(* POU Simulation/FB_Simu_Manipulator, ST *)
FUNCTION_BLOCK FB_Simu_Manipulator
(*Simulation model for the behaviour of the Manipulator.
Author: Niko Siltala, niko.siltala@tut.fi, Tampere University of Technology / MEI
Date: 2016-12-12
Version: 1.0
*)
VAR_INPUT
	bEnable			: BOOL := TRUE;	(*Enable manipulator*)
	bLift_Start		: BOOL;	(*Triggers and starts the lift movement at rising edge*)
	fLift_Velo		: REAL := 10;	(*Velocity*)
	fLift_TargetPos	: REAL;	(*Target position*)
	bBeam_Left		: BOOL;	(*Turn beam at left*)
	bBeam_Right		: BOOL;	(*Turn beam at right*)
	bGripper_Close	: BOOL; (*Close Gripper*)
END_VAR
VAR_OUTPUT
	bGripperIsOpen	: BOOL;	(*Gripper is open*)
	bLift_InTarget	: BOOL;	(*Lift has reached the target*)
	fLift_CurrentPos	: REAL;	(*Current position of the lift*)
	bLimit_Top		: BOOL;	(*Height position at top limit*)
	bLimit_Bottom	: BOOL;	(*Height position at bottom limit*)
	bHome_Sensor	: BOOL;	(*Height position at home limit*)
	bBeamAtRight	: BOOL;	(*Beam turned into right limit*)
	bBeamAtLeft		: BOOL;	(*Beam turned into left limit*)
END_VAR
VAR_IN_OUT
	stPart_inGripper : ST_Part; 	(*Data structure for the part*)
END_VAR
VAR
	fPos_angle	: REAL := 70;	(*Angle of beam [deg]*)
	fPos_height	: REAL;	(* Manipulators height position*)
	fPos_X		: REAL;	(* Manipulator's X position*)
	fPos_Y		: REAL;	(* Manipulator's Y position*)
	fBasePos_Y 	: REAL; (*Position of manipulator base*)
	iState_Lift		: UINT;	(*State of beam model*)
	fPos_Beam_L	: REAL;	(*Beam position left end*)
	fPos_Beam_R	: REAL;	(*Beam position right end*)
	bGripperClosed	: BOOL; (*Gripper is closed*)
	fPosFingerDiff 	: REAL;	(*Right finger position. 0 poistion when grasping.*)
	bInitDone		: BOOL;		(*Initialisation done for simulated machine*)
END_VAR
VAR CONSTANT
	iBEAM_LENGTH	: USINT := 120;	(*length of the beam*)
	fPOS_MAX_DOWN	: REAL	:= 220;	(*Max position for down movement*)
END_VAR
(*Simulate axis*)
IF NOT bEnable THEN
	iState_Lift := 0;
END_IF;

(*Initialisation*)
IF NOT bInitDone THEN
	(*Randomize system's starting position*)
	lastRandom := RDM(lastRandom);
	fLift_CurrentPos := -100 * lastRandom + 10;
	lastRandom := RDM(lastRandom);
	fPos_angle := 100 * lastRandom + 40; (* X2 = (180 - 100[=X1]) / 2 *)
	bInitDone:=TRUE;
END_IF;

CASE iState_Lift OF
0:	(*Off*)
	IF bEnable THEN
		iState_Lift := 1;
	ELSE
		bLift_InTarget := FALSE;
	END_IF;

1:	(*IDLE*)
	IF bLift_Start THEN
		bLift_InTarget := FALSE;
		iState_Lift := 2;
	END_IF;

2:	(*MovingToTarget*)
	bLift_InTarget := FALSE;
	IF fLift_TargetPos > fLift_CurrentPos THEN
		(*Moving up*)
		fLift_CurrentPos := fLift_CurrentPos + ABS(fLift_Velo);
	ELSIF fLift_TargetPos < fLift_CurrentPos THEN
		(*Moving down*)
		fLift_CurrentPos := fLift_CurrentPos - ABS(fLift_Velo);
	END_IF;
	(*Limit output*)
	fLift_CurrentPos := LIMIT(-220, fLift_CurrentPos, 10);
	(* Moved close to target*)
	IF (ABS(fLift_CurrentPos - fLift_TargetPos) <= ABS(fLift_Velo) ) THEN
		fLift_CurrentPos := fLift_TargetPos;
		iState_Lift := 3;
	END_IF;
	(*Start has been removed*)
	IF NOT bLift_Start THEN
		iState_Lift := 1;
	END_IF;

3:	(*In target*)
	bLift_InTarget := TRUE;
	IF NOT bLift_Start THEN
		iState_Lift := 1;
	END_IF;

ELSE	(*Error / to Default*)
	iState_Lift := 0;
END_CASE;

fPos_Y := -fLift_CurrentPos;


(*Simulate Beam turning*)
IF bBeam_Left AND (fPos_angle > 0) AND NOT bBeam_Right THEN
	fPos_angle := LIMIT(0, (fPos_angle - 15), 180);
END_IF;
IF bBeam_Right AND (fPos_angle < 180) AND NOT bBeam_Left THEN
	fPos_angle := LIMIT(0, (fPos_angle + 15), 180);
END_IF;


(*Calculate visualisation positions for lift and beam*)
fPos_X := -iBEAM_LENGTH*COS(3.1415926535897932384626433832795/180*fPos_angle);
(*fPos_Y := fPos_height;*)
fBasePos_Y := fPos_Y;	(*Used for animations as base position*)

(*Calculate endpositions of the visualisation for the beam*)
IF (fPos_X > 0) THEN
	fPos_Beam_L := 0;
	fPos_Beam_R := fPos_X;
ELSE
	fPos_Beam_L := fPos_X;
	fPos_Beam_R := 0;
END_IF;

(*define finger positions*)
IF bGripper_Close THEN
	fPosFingerDiff := 0;
ELSE
	fPosFingerDiff := 10;
END_IF;

(*Set sensor values*)
(*Set output values*)
bLimit_Top := (fPos_Y <= 0);
bLimit_Bottom := (fPos_Y >= 210);
bHome_Sensor := (fPos_Y <= 5) AND (fPos_Y >= -5);

bBeamAtLeft := (fPos_angle <= 0);
bBeamAtRight := (fPos_angle >= 180);

bGripperIsOpen := NOT bGripper_Close;
bGripperClosed := bGripper_Close;
END_FUNCTION_BLOCK

(* POU Simulation/RDM_From_OSCAT/RDM, ST *)
FUNCTION RDM : REAL
VAR_INPUT
	last : REAL;
END_VAR
VAR
	tn : DWORD;
	tc : INT;
END_VAR
(*
FROM OSCAT 333
version 1.9	10. mar. 2009
programmer 	hugo
tested by		tobias

this function calculates a pseudo random number
to generate the number it reads the sps timer and calculates a random number between 0 and 1:
in order to use rdm more then once within one sps cycle it need to be called with different seed numbers LAST.

*)
tn := T_PLC_MS();
tc := BIT_COUNT(tn);
tn.31 := tn.2;
tn.30 := tn.5;
tn.29 := tn.4;
tn.28 := tn.1;
tn.27 := tn.0;
tn.26 := tn.7;
tn.25 := tn.6;
tn.24 := tn.3;
tn := ROL(tn,BIT_COUNT(tn)) OR 16#80000001;
tn := tn MOD 71474513 + INT_TO_DWORD(tc + 77);
RDM := FRACT(DWORD_TO_REAL(tn) / 10000000.0 * (math.E - LIMIT(0.0,last,1.0)));


(*
pt := ADR(temp);
pt^ := (T_PLC_MS() AND 16#007FFFFF) OR 16#3D000000;
RDM := fract(modR(temp*e+pi1, PI1-last) + modR(temp*PI1+e + last,e-last));
*)

(* revision history
hm		16. jan 2007		rev 1.0
	original version

hm		11. nov 2007		rev 1.1
	changed time() into t_plc_ms()

hm		20. nov 2007		rev 1.2
	changed code of temp calculation to avoid overflow in modr due to resuclt would not fit DINT for high timeer values

hm		5. jan 2008		rev 1.3
	changed calculation of temp to avoid problem with high values of t_plc_ms

hm		2. feb 2008		rev 1.4
	changed algorithm to avoind non iec functions and guarantee more randomness

hm	10. mar. 2008		rev 1.5
	make sure last will be between 0 and 1 to avoid invalid results

hm	16. mar. 2008		rev 1.6
	added conversion for tc to avoid warnings under codesys 3.0

hm	18. may. 2008		rev 1.7
	changed constant E to E1

hm	18. oct. 2008		rev 1.8
	using math constants

hm	10. mar. 2009		rev 1.9
	real constants updated to new systax using dot

*)
END_FUNCTION

(* POU Simulation/RDM_From_OSCAT/T_PLC_MS, ST *)
FUNCTION T_PLC_MS : DWORD
VAR CONSTANT
	debug : BOOL := 0;
	N : INT := 0;
	offset : DWORD := 0;
END_VAR
VAR
	tx : TIME;
END_VAR
(*
	From OSCAT 333
	version 1.2	16. nov 2008
	programmer 	hugo
	tested BY	oscat

	T_PLC_MS reads the internal PLC timer AND RETURN the TIME, it has the advantage TO be able TO set a debug mode
AND SPEED up the counter TO test the plc timer overrun which occurs every 50 days respectively 25 days AT siemens S7
	this routine also allows TO correct the behavior OF s7 where the internal plc counter will NOT count all 32 bits.
*)
tx := TIME();
T_PLC_MS := TIME_TO_DWORD(Tx);
(* hier muss die korrektur für step7 stattfinden
plctime muss den vollen wertebereich von time ausnutzen:
wenn bei step7 time -24tage bis plus 24 tage ist dann muss der timer auch beim überlauf auf -24tage springen 
und auf keinen fall auf 0 !!!!
für siemens muss ein weiterer fb im main eingebunden werden der sicherstellt das alle 32 bits durchgezählt werden.
es kann nur ein fb sein den er muss sich das oberste (32te) bit merken.
oder etwa spring s7 bei überlauf auf -24 tage????? dann wäre keine korrektur nötig.
*)
IF debug THEN
	T_PLC_MS := (SHL(T_PLC_MS,N) OR SHL(DWORD#1,N)-1) + OFFSET;
END_IF;

(* revision history
hm	14.9.2007	rev 1.0
	original version

hm	12. nov 2007	rev 1.1
	added temporaray variable tx because some compilers could not handle time() as an argument

hm	16. nov. 2008	rev 1.2
	initialized constants with 0 for compatibility reasons
*)
END_FUNCTION

(* POU Simulation/RDM_From_OSCAT/BIT_COUNT, ST *)
FUNCTION BIT_COUNT : INT
VAR_INPUT
	IN : DWORD;
END_VAR
VAR
END_VAR
(*
OSCAT 333
version 1.1	10 sep 2007
programmer 	hugo
tested by		tobias

BIT_COUNT counts the amount True of bits in a dword.
for exabple: bit_count(3) returns 2 because two bits (bits 0 and 1) are true and all others are false. 
*)
WHILE in > 0 DO
	IF in.0 THEN Bit_Count := Bit_Count + 1; END_IF;
	in := SHR(in,1);
END_WHILE;



(* revision history
5.7.2007	rev 1.0		original version

10.9.2007	rev 1.1		hm
	changed algorithm for better performace
	the execution time has reduced by a factor of 5
	deleted unused variable temp
*)
END_FUNCTION

(* POU Simulation/RDM_From_OSCAT/FRACT, ST *)
FUNCTION FRACT : REAL
VAR_INPUT
	x : REAL;
END_VAR
VAR
END_VAR
(*
From OSCAT 333
version 1.3	10. mar. 2009
programmer 	hugo
tested by		tobias

this function returns the fraction of a real number
fract(3.14) = 0.14

*)
IF ABS(x) < 2.0E9 THEN
	FRACT := x - DINT_TO_REAL(D_TRUNC(x));
ELSE
	FRACT := 0.0;
END_IF;

(* revision history
hm	4. aug 2006	rev 1.0
	original version

hm	11. mar 2008	rev 1.1
	added dint_to_real for compatibility reasons
	now returns 0 for number > 2e9
	changed input to x

hm	21. mar. 2008	rev 1.2
	use D_trunc instead of TRUNC for compatibility reasons

hm	10. mar. 2009	rev 1.3
	real constants updated to new systax using dot

*)
END_FUNCTION

(* POU Simulation/RDM_From_OSCAT/D_TRUNC, ST *)
FUNCTION D_TRUNC : DINT
VAR_INPUT
	X : REAL;
END_VAR
VAR
END_VAR
(*
From OSCAT 333
version 1.2	10. mar. 2009
programmer 	hugo
tested by		oscat

d_trunc truncates a real to a dint 1.5 will be 1 and -1.5 will be -1
d_trunc is necessary because many systems do not offer a trunc to a dint
also real_to_dint will not deliver the same result on different systems

*)
D_TRUNC := REAL_TO_DINT(X);
IF X > 0.0 THEN
	IF DINT_TO_REAL(D_TRUNC) > X THEN D_TRUNC := D_TRUNC - 1; END_IF;
ELSE
	IF DINT_TO_REAL(D_TRUNC) < X THEN D_TRUNC := D_TRUNC + 1; END_IF;
END_IF;


(* for systems that support a dint truncation this routine can be replaced by trunc() *)


(* revision history
hm	21. mar. 2008	rev 1.0
	original version

hm	31. oct. 2008	rev 1.1
	optimized performance

hm	10. mar. 2009	rev 1.2
	real constants updated to new systax using dot
*)
END_FUNCTION

(* POU Simulation/FB_Simu_Drill, ST *)
FUNCTION_BLOCK FB_Simu_Drill
(*Simulation model for the behaviour of the Drill machine.
Author: Niko Siltala, niko.siltala@tut.fi, Tampere University of Technology / MEI
Date: 2016-12-12
Version: 1.0
*)
VAR_INPUT
	bEnable			: BOOL := TRUE;	(*Enable drill*)
	bLift_Start		: BOOL;		(*Triggers and starts the lift movement at rising edge*)
	fLift_Velo		: REAL := 10;	(*Velocity*)
	fLift_TargetPos	: REAL;		(*Target position*)
	bDrillOn			: BOOL;		(*Drill is On*)
	bFixture_Close	: BOOL; 	(*Close Fixture*)
	bInitDone		: BOOL;		(*Initialisation done for simulated machine*)
END_VAR
VAR_OUTPUT
	bLift_InTarget	: BOOL;	(*Lift has reached the target*)
	fLift_CurrentPos	: REAL;	(*Current position of the lift*)
	bLimit_Top		: BOOL;	(*Height position at top limit*)
	bLimit_Bottom	: BOOL;	(*Height position at bottom limit*)
	bHome_Sensor	: BOOL;	(*Height position at home limit*)
	bFixture_Open	: BOOL;	(*Fixture is Open*)
	bFixture_Closed	: BOOL;	(*Fixture is Closed*)
END_VAR
VAR_IN_OUT
	stPart_inFixture : ST_Part; 	(*Data structure for the part*)
END_VAR
VAR
	fPos_height	: REAL;	(* Manipulators height position*)
	fPos_Y		: REAL;	(* Manipulator's Y position*)
	fBasePos_Y 	: REAL; (*Position of manipulator base*)
	iState_Lift	: UINT;	(*State of beam model*)
	iRPMCurrent	: INT;	(*Current RPM*)
	fPosJawDiff 	: REAL;	(*Right fixture jaw position. 0 position when grasping.*)
END_VAR
VAR CONSTANT
	fPOS_MAX_DOWN		: REAL	:= 170;	(*Max position for down movement*)
	iSPINDLE_RPM_MAX	: INT	:= 600;	(*Max RPM for Spindle*)
END_VAR
(*Simulate axis*)
IF NOT bEnable THEN
	iState_Lift := 0;
END_IF;

(*Initialisation*)
IF NOT bInitDone THEN
	(*Randomize system's starting position*)
	lastRandom := RDM(lastRandom);
	fLift_CurrentPos := -60 * lastRandom + 10;
	bInitDone:=TRUE;
END_IF;

CASE iState_Lift OF
0:	(*Off*)
	IF bEnable THEN
		iState_Lift := 1;
	ELSE
		bLift_InTarget := FALSE;
	END_IF;

1:	(*IDLE*)
	IF bLift_Start THEN
		bLift_InTarget := FALSE;
		iState_Lift := 2;
	END_IF;

2:	(*MovingToTarget*)
	bLift_InTarget := FALSE;
	IF fLift_TargetPos > fLift_CurrentPos THEN
		(*Moving up*)
		fLift_CurrentPos := fLift_CurrentPos + ABS(fLift_Velo);
	ELSIF fLift_TargetPos < fLift_CurrentPos THEN
		(*Moving down*)
		fLift_CurrentPos := fLift_CurrentPos - ABS(fLift_Velo);
	END_IF;
	(*Limit output*)
	fLift_CurrentPos := LIMIT(-fPOS_MAX_DOWN, fLift_CurrentPos, 10);
	(* Moved close to target*)
	IF (ABS(fLift_CurrentPos - fLift_TargetPos) <= ABS(fLift_Velo) ) THEN
		fLift_CurrentPos := fLift_TargetPos;
		iState_Lift := 3;
	END_IF;
	(*Start has been removed*)
	IF NOT bLift_Start THEN
		iState_Lift := 1;
	END_IF;

3:	(*In target*)
	bLift_InTarget := TRUE;
	IF NOT bLift_Start THEN
		iState_Lift := 1;
	END_IF;

ELSE	(*Error / to Default*)
	iState_Lift := 0;
END_CASE;

fPos_Y := -fLift_CurrentPos;
fBasePos_Y := fPos_Y;	(*Used for animations as base position*)


(*define fixture jaws positions*)
IF bFixture_Close THEN
	fPosJawDiff := 0;
ELSE
	fPosJawDiff := 10;
END_IF;

(*Set sensor values*)
(*Set output values*)
bLimit_Top := (fPos_Y <= 0);
bLimit_Bottom := (fPos_Y >= (fPOS_MAX_DOWN-10));
bHome_Sensor := (fPos_Y <= 5) AND (fPos_Y >= -5);

bFixture_Open := NOT bFixture_Close;
bFixture_Closed := bFixture_Close;

IF bDrillOn THEN
	iRPMCurrent := iRPMCurrent + 100;
ELSE
	iRPMCurrent := iRPMCurrent - 20;
END_IF;
iRPMCurrent := LIMIT(0, iRPMCurrent, iSPINDLE_RPM_MAX);
END_FUNCTION_BLOCK

(* POU Simulation/F_MovePartForward, ST *)
FUNCTION F_MovePartForward : BOOL
(*Moves parts forward on conveyour, if possible*)
VAR_INPUT
END_VAR
VAR_IN_OUT
	arrParts : ARRAY [0..10] OF ST_Part;	(*Array of parts*)
END_VAR
VAR
	i : INT;	(*indexer*)
	j : INT;	(*indexer*)
END_VAR
(*Moves parts forward as much there is free places*)
FOR i:= 0 TO 9 DO
	j := i +1;
	IF NOT arrParts[i].bExists THEN
		IF arrParts[j].bExists THEN
			F_CopyPart(arrParts[j], arrParts[i]);
			arrParts[j].bExists := FALSE;
			arrParts[j].bHasHole := FALSE;
		END_IF;
	END_IF;
END_FOR;

F_MovePartForward := TRUE;
END_FUNCTION

(* POU Simulation/F_CopyPart, ST *)
FUNCTION F_CopyPart : BOOL
(*Moves part data from part to part*)
VAR_INPUT
END_VAR
VAR_IN_OUT
	stPartFrom : ST_Part;	(*The copied part - From*)
	stPartTo : ST_Part;	(*Where to copy the part*)
END_VAR
VAR
END_VAR
(*Moves part data from part to part*)
stPartTo.bExists := stPartFrom.bExists;
stPartTo.bHasHole := stPartFrom.bHasHole;
stPartTo.posX := stPartFrom.posX;
stPartTo.posY := stPartFrom.posY;

F_CopyPart:=TRUE;
END_FUNCTION

(* POU Examples/FB_SFC_Example, SFC *)
FUNCTION_BLOCK FB_SFC_Example
VAR_INPUT
	bReset		: BOOL;	(*Reset Request*)
END_VAR
VAR_OUTPUT
END_VAR
VAR
	bLocalReset	: BOOL;	(*Performs local reset*)
	SFCReset 	: BOOL;	(*Resets the execution of SFC to init once this SFCFlag is set true *)
END_VAR
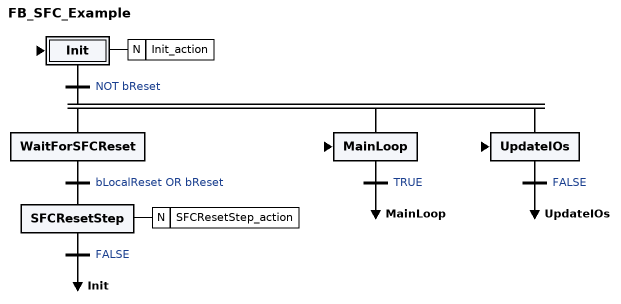
INITIAL_STEP Init:
	Init_action(N);
END_STEP
TRANSITION FROM Init TO (WaitForSFCReset, MainLoop, UpdateIOs) := NOT bReset;
END_TRANSITION
STEP WaitForSFCReset:
END_STEP
TRANSITION FROM WaitForSFCReset TO SFCResetStep := bLocalReset OR bReset;
END_TRANSITION
STEP MainLoop:
END_STEP
TRANSITION FROM MainLoop TO MainLoop := TRUE;
END_TRANSITION
STEP UpdateIOs:
END_STEP
TRANSITION FROM UpdateIOs TO UpdateIOs := FALSE;
END_TRANSITION
STEP SFCResetStep:
	SFCResetStep_action(N);
END_STEP
TRANSITION FROM SFCResetStep TO Init := FALSE;
END_TRANSITION

ACTION Init_action:
SFCReset := FALSE;
bLocalReset	:= FALSE;
END_ACTION

ACTION SFCResetStep_action:
SFCReset := TRUE;
END_ACTION
END_FUNCTION_BLOCK

(* POU Examples/FB_SimpleManager, ST *)
FUNCTION_BLOCK FB_SimpleManager
(*Simple manager following emergency and run/stop state. Outputs can be used to enable user's processes and programs.
Niko Siltala niko.siltala@tuni.fi, 
Tampere University, ENS, ATME.
9.10.2019 v1 *)
VAR_INPUT
	bEmergencyClear	: BOOL;	(*Emergency cleared*)
	bReset				: BOOL;	(*Reset signal*)
	bStart				: BOOL;	(*Start signal*)
	bStop				: BOOL;	(*Stop signal*)
END_VAR
VAR_OUTPUT
	oEmergencyClear	: BOOL;	(*Emergency is cleared*)
	oRun				: BOOL;	(*System can be started and running*)
END_VAR
VAR
	rsEmergency	: RS;
	rsRunning		: RS;
	bResetRequired	: BOOL := TRUE;	(*reset is required*)
END_VAR
(*Defaults*)

(*Reset done*)
IF bReset THEN
	bResetRequired	:= FALSE;
END_IF;

(*Emergency active or cleared?*)
rsEmergency(
	SET:= bReset,
	RESET1:= NOT bEmergencyClear,
	Q1=> oEmergencyClear );

(*Running or stop?*)
rsRunning(
	SET:= bStart,
	RESET1:= (NOT oEmergencyClear) OR bStop OR bResetRequired,
	Q1=> oRun );
END_FUNCTION_BLOCK

(* POU Examples/FB_SimpleModeManager, ST *)
FUNCTION_BLOCK FB_SimpleModeManager
(*Simple manager following emergency and run/stop state. Implemented through state model.
Includes manager for two control modes. Outputs can be used to enable user's processes and programs.
Niko Siltala niko.siltala@tuni.fi, 
Tampere University, ENS, ATME.
9.10.2019 v1 *)
VAR_INPUT
	bEmergencyClear	: BOOL;	(*Emergency cleared*)
	bReset				: BOOL;	(*Reset signal*)
	bStart				: BOOL;	(*Start signal*)
	bStop				: BOOL;	(*Stop signal*)
	bSelectMode_Auto	: BOOL;	(*Mode select request : Auto *)
	bSelectMode_Manu	: BOOL;	(*Mode select request : Manual *)
END_VAR
VAR_OUTPUT
	oEmergencyClear	: BOOL;	(*Emergency is cleared*)
	oRun				: BOOL;	(*System can be started and running*)
	oModeAct_Auto		: BOOL;	(*Mode active : Auto *)
	oModeAct_Manu	: BOOL;	(*Mode active : Manual *)
	oModeAct			: EN_Mode;	(*Current active mode*)
END_VAR
VAR
	modePrev		: EN_Mode;			(*Mode at previous PLC cycle*)
	bModeChanged	: BOOL;			(*Mode has changed*)
	bResetRequired	: BOOL := TRUE;	(*reset is required*)
	iState			: INT := 0;			(*State*)
END_VAR
(*Default values for each PLC cycle*)
bModeChanged := FALSE;
oModeAct_Auto := FALSE;
oModeAct_Manu := FALSE;

(****** SECTION: INPUTS PROCESSING ******)
(*Update current control mode*)
IF bSelectMode_Auto THEN
	oModeAct := eMode_Auto;
ELSIF bSelectMode_Manu THEN
	oModeAct := eMode_Manual;
END_IF;

(*Observe mode change request*)
IF oModeAct <> modePrev THEN
	modePrev := oModeAct;
	bModeChanged := TRUE;
	bResetRequired	:= TRUE;
END_IF;

(****** SECTION: STATE MODEL ******)
(*Emergency is active. Force state to emergency active*)
IF NOT bEmergencyClear THEN
	iState := 0;
END_IF;

(*State model*)
CASE iState  OF
0:	(*Emergency active*)
	IF bReset AND bEmergencyClear THEN
		iState := 10;
	END_IF;

10: (*Reset required *)
	IF bReset THEN
		iState := 12;
		bResetRequired	:= FALSE;
	END_IF;

12:	(*Stopped*)
	IF bResetRequired THEN
		iState := 10;
	ELSIF bStart AND NOT bStop THEN
		iState := 20;
	END_IF;

20: (*Run / Running*)
	IF bResetRequired OR bModeChanged THEN
		iState := 10;
	ELSIF bStop THEN
		iState := 12;
	END_IF;

ELSE	(*Default state*)
	iState := 0;
END_CASE;

(****** SECTION: OUTPUTS ******)
(*Set manager outputs according the state*)
oEmergencyClear := (iState>0);
oRun := (iState>=20);

(*Update binary outputs for Control Modes*)
CASE oModeAct  OF
eMode_Auto:
	oModeAct_Auto:= TRUE;
eMode_Manual:
	oModeAct_Manu := TRUE;
END_CASE;
END_FUNCTION_BLOCK

(* POU Examples/FB_SimpleModeManager2, ST *)
FUNCTION_BLOCK FB_SimpleModeManager2
(*Simple manager following emergency and run/stop state. Includes manager for two control modes. Implemented with FBDs.
Outputs can be used to enable user's processes and programs.
Niko Siltala niko.siltala@tuni.fi, 
Tampere University, ENS, ATME.
9.10.2019 v1 *)
VAR_INPUT
	bEmergencyClear	: BOOL;	(*Emergency cleared*)
	bReset				: BOOL;	(*Reset signal*)
	bStart				: BOOL;	(*Start signal*)
	bStop				: BOOL;	(*Stop signal*)
	bSelectMode_Auto	: BOOL;	(*Mode select request : Auto *)
	bSelectMode_Manu	: BOOL;	(*Mode select request : Manual *)
END_VAR
VAR_OUTPUT
	oEmergencyClear	: BOOL;	(*Emergency is cleared*)
	oRun				: BOOL;	(*System can be started and running*)
	oModeAct_Auto		: BOOL;	(*Mode active : Auto *)
	oModeAct_Manu	: BOOL;	(*Mode active : Manual *)
	oModeAct			: EN_Mode;	(*Current active mode*)
END_VAR
VAR
	rsEmergency	: RS;
	rsRunning		: RS;
	modePrev		: EN_Mode;			(*Mode at previous PLC cycle*)
	bModeChanged	: BOOL;			(*Mode has changed*)
	bResetRequired	: BOOL := TRUE;	(*reset is required*)
END_VAR
(*Default values for each PLC cycle*)
bModeChanged := FALSE;
oModeAct_Auto := FALSE;
oModeAct_Manu := FALSE;

(*Reset done*)
IF bReset THEN
	bResetRequired	:= FALSE;
END_IF;

(*Update current control mode*)
IF bSelectMode_Auto THEN
	oModeAct := eMode_Auto;
ELSIF bSelectMode_Manu THEN
	oModeAct := eMode_Manual;
END_IF;

(*Observe mode change request*)
IF oModeAct <> modePrev THEN
	modePrev := oModeAct;
	bModeChanged := TRUE;
	bResetRequired	:= TRUE;
END_IF;

(*Calling action containing FBD code for deciding emergency and run output states*)
act_fbd_controls();

(*Update binary outputs for Control Modes*)
CASE oModeAct  OF
eMode_Auto:
	oModeAct_Auto:= TRUE;
eMode_Manual:
	oModeAct_Manu := TRUE;
END_CASE;
END_FUNCTION_BLOCK
ACTION act_fbd_controls:
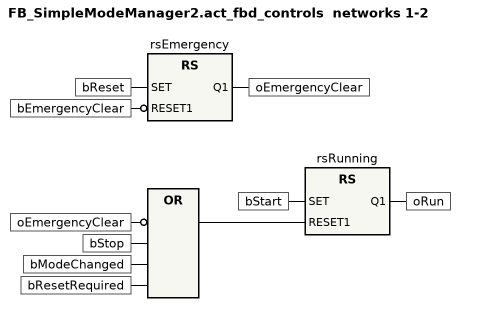
_FBD_ (* Function Block Diagram *)
NETWORK 1
	rsEmergency:RS(SET: bReset, RESET1: NOT bEmergencyClear) => oEmergencyClear
NETWORK 2
	rsRunning:RS(SET: bStart, RESET1: OR(NOT oEmergencyClear, bStop, bModeChanged, bResetRequired)) => oRun
_END_FBD_
(* the same logic as Structured Text *)
(* Network 1 *)
rsEmergency(SET := bReset, RESET1 := NOT bEmergencyClear);
oEmergencyClear := rsEmergency.Q1;
(* Network 2 *)
rsRunning(SET := bStart, RESET1 := NOT oEmergencyClear OR bStop OR bModeChanged OR bResetRequired);
oRun := rsRunning.Q1;
END_ACTION

(* Visualisation Simulator/Components/VC_Beacon
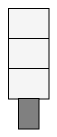
rectangle at (0,0)-(41,31): alarm colour if $red$
rectangle at (0,30)-(41,61): alarm colour if $yellow$
rectangle at (0,60)-(41,91): alarm colour if $green$
1 more shapes without text or variables
*)

(* Visualisation Simulator/ErrorPanels/VC_ErrorDetail_Drill
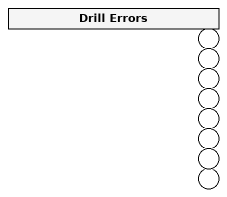
embedded screen at (0,20)-(211,41): VC_ErrorItem
rectangle at (0,0)-(211,21): text "Drill Errors"
embedded screen at (0,40)-(211,61): VC_ErrorItem
embedded screen at (0,160)-(211,181): VC_ErrorItem
embedded screen at (0,60)-(211,81): VC_ErrorItem
embedded screen at (0,80)-(211,101): VC_ErrorItem
embedded screen at (0,100)-(211,121): VC_ErrorItem
embedded screen at (0,120)-(211,141): VC_ErrorItem
embedded screen at (0,140)-(211,161): VC_ErrorItem
*)

(* Visualisation Simulator/ErrorPanels/VC_ErrorDetail_Manip
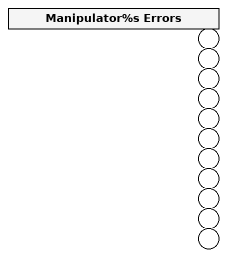
embedded screen at (0,20)-(211,41): VC_ErrorItem
rectangle at (0,0)-(211,21): text "Manipulator%s Errors"; shows $manipName$
embedded screen at (0,40)-(211,61): VC_ErrorItem
embedded screen at (0,60)-(211,81): VC_ErrorItem
embedded screen at (0,80)-(211,101): VC_ErrorItem
embedded screen at (0,80)-(211,101): VC_ErrorItem
embedded screen at (0,100)-(211,121): VC_ErrorItem
embedded screen at (0,120)-(211,141): VC_ErrorItem
embedded screen at (0,140)-(211,161): VC_ErrorItem
embedded screen at (0,160)-(211,181): VC_ErrorItem
embedded screen at (0,180)-(211,201): VC_ErrorItem
embedded screen at (0,200)-(211,221): VC_ErrorItem
embedded screen at (0,220)-(211,241): VC_ErrorItem
*)

(* Visualisation Simulator/VC_ErrorDetails
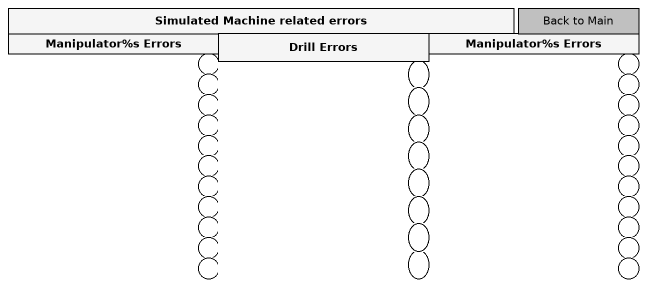
embedded screen at (0,25)-(211,271): VC_ErrorDetail_Manip
rectangle at (0,0)-(506,26): text "Simulated Machine related errors"
embedded screen at (420,25)-(631,271): VC_ErrorDetail_Manip
embedded screen at (210,25)-(421,271): VC_ErrorDetail_Drill
rounded rectangle at (510,0)-(631,26): text "Back to Main"; opens VISU_SimulatedMachine
*)

(* Visualisation Simulator/Components/VC_ErrorItem
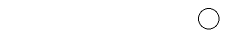
rectangle at (0,0)-(191,21): text "%s :"; shows $name$; alarm colour if $flag$
ellipse at (190,0)-(211,21): alarm colour if $flag$
1 more shapes without text or variables
*)

(* Visualisation Simulator/FBs/VC_FB_Simu_Drill
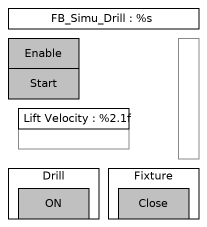
rectangle at (100,160)-(191,211): text "Fixture"
rectangle at (0,160)-(91,211): text "Drill"
rounded rectangle at (0,30)-(71,61): text "Enable"; alarm colour if $FB$.bEnable; toggles $FB$.bEnable
rectangle at (0,0)-(191,21): text "FB_Simu_Drill : %s"; shows $Name$
rounded rectangle at (0,60)-(71,91): text "Start"; alarm colour if $FB$.bLift_Start; taps $FB$.bLift_Start
rectangle at (10,100)-(121,121): text "Lift Velocity : %2.1f"; shows $FB$.fLift_Velo
rounded rectangle at (10,180)-(81,211): text "ON"; alarm colour if $FB$.bDrillOn; toggles $FB$.bDrillOn
rounded rectangle at (110,180)-(181,211): text "Close"; alarm colour if $FB$.bFixture_Close; toggles $FB$.bFixture_Close
2 more shapes without text or variables
1 elements of other kinds (tables, trends, ...) not read
*)

(* Visualisation Simulator/FBs/VC_FB_Simu_Manipulator
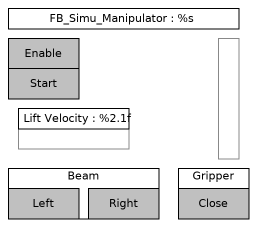
rectangle at (170,160)-(241,211): text "Gripper"
rectangle at (0,160)-(151,211): text "Beam"
rounded rectangle at (0,30)-(71,61): text "Enable"; alarm colour if $FB$.bEnable; toggles $FB$.bEnable
rectangle at (0,0)-(231,21): text "FB_Simu_Manipulator : %s"; shows $Name$
rounded rectangle at (0,60)-(71,91): text "Start"; alarm colour if $FB$.bLift_Start; taps $FB$.bLift_Start
rectangle at (10,100)-(121,121): text "Lift Velocity : %2.1f"; shows $FB$.fLift_Velo
rounded rectangle at (0,180)-(71,211): text "Left"; alarm colour if $FB$.bBeam_Left; toggles $FB$.bBeam_Left
rounded rectangle at (80,180)-(151,211): text "Right"; alarm colour if $FB$.bBeam_Right; toggles $FB$.bBeam_Right
rounded rectangle at (170,180)-(241,211): text "Close"; alarm colour if $FB$.bGripper_Close; toggles $FB$.bGripper_Close
2 more shapes without text or variables
1 elements of other kinds (tables, trends, ...) not read
*)

(* Visualisation Visual Components/VC_PackMLStates
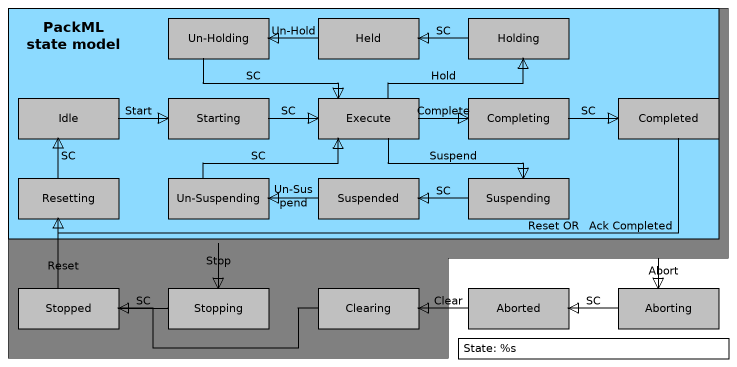
rounded rectangle at (160,280)-(261,321): text "Stopping"; alarm colour if $PackML$.eState = 4
rounded rectangle at (10,90)-(111,131): text "Idle"; alarm colour if $PackML$.eState = 6
rounded rectangle at (160,170)-(261,211): text "Un-Suspending"; alarm colour if $PackML$.eState = 11
rounded rectangle at (610,280)-(711,321): text "Aborting"; alarm colour if $PackML$.eState = 0
rounded rectangle at (460,280)-(561,321): text "Aborted"; alarm colour if $PackML$.eState = 1
rectangle at (450,330)-(721,351): text "State: %s"; shows $PackML$.strState
rounded rectangle at (310,280)-(411,321): text "Clearing"; alarm colour if $PackML$.eState = 2
rounded rectangle at (10,280)-(111,321): text "Stopped"; alarm colour if $PackML$.eState = 3
rounded rectangle at (10,170)-(111,211): text "Resetting"; alarm colour if $PackML$.eState = 5
rounded rectangle at (160,90)-(261,131): text "Starting"; alarm colour if $PackML$.eState = 7
rounded rectangle at (310,90)-(411,131): text "Execute"; alarm colour if $PackML$.eState = 8
rounded rectangle at (460,90)-(561,131): text "Completing"; alarm colour if $PackML$.eState = 15
rounded rectangle at (610,90)-(711,131): text "Completed"; alarm colour if $PackML$.eState = 16
rounded rectangle at (310,170)-(411,211): text "Suspended"; alarm colour if $PackML$.eState = 10
rounded rectangle at (460,170)-(561,211): text "Suspending"; alarm colour if $PackML$.eState = 9
rounded rectangle at (460,10)-(561,51): text "Holding"; alarm colour if $PackML$.eState = 12
rounded rectangle at (310,10)-(411,51): text "Held"; alarm colour if $PackML$.eState = 13
rounded rectangle at (160,10)-(261,51): text "Un-Holding"; alarm colour if $PackML$.eState = 14
polyline at (645,250)-(655,280): alarm colour if $PackML$.bAbort
rectangle at (635,255)-(676,271): text "Abort"; alarm colour if $PackML$.bAbort
polyline at (205,235)-(215,280): alarm colour if $PackML$.bStop
rectangle at (190,245)-(231,261): text "Stop"; alarm colour if $PackML$.bStop
polyline at (195,130)-(335,170): alarm colour if $PackML$.bSC
rectangle at (235,140)-(266,156): text "SC"; alarm colour if $PackML$.bSC
polyline at (195,50)-(335,90): alarm colour if $PackML$.bSC
polyline at (380,50)-(520,90): alarm colour if $PackML$.bHold
rectangle at (420,60)-(451,76): text "Hold"; alarm colour if $PackML$.bHold
polyline at (560,295)-(610,305): alarm colour if $PackML$.bSC
polyline at (45,210)-(55,280): alarm colour if $PackML$.bReset
polyline at (110,105)-(160,115): alarm colour if $PackML$.bStart
polyline at (110,295)-(310,340): alarm colour if $PackML$.bSC
rectangle at (230,60)-(261,76): text "SC"; alarm colour if $PackML$.bSC
polyline at (380,130)-(520,170): alarm colour if $PackML$.bSuspend
rectangle at (415,140)-(476,156): text "Suspend"; alarm colour if $PackML$.bSuspend
rectangle at (120,285)-(151,301): text "SC"; alarm colour if $PackML$.bSC
rectangle at (570,285)-(601,301): text "SC"; alarm colour if $PackML$.bSC
polyline at (410,295)-(460,305): alarm colour if $PackML$.bClear
rectangle at (420,285)-(461,301): text "Clear"; alarm colour if $PackML$.bClear
polyline at (260,105)-(310,115): alarm colour if $PackML$.bSC
rectangle at (265,95)-(296,111): text "SC"; alarm colour if $PackML$.bSC
rectangle at (110,95)-(151,111): text "Start"; alarm colour if $PackML$.bStart
rectangle at (35,250)-(76,266): text "Reset"; alarm colour if $PackML$.bReset
polyline at (410,185)-(460,195): alarm colour if $PackML$.bSC
rectangle at (420,175)-(451,191): text "SC"; alarm colour if $PackML$.bSC
polyline at (410,25)-(460,35): alarm colour if $PackML$.bSC
rectangle at (420,15)-(451,31): text "SC"; alarm colour if $PackML$.bSC
polyline at (260,185)-(310,195): alarm colour if $PackML$.bUn_Suspend
rectangle at (260,170)-(311,206): text "Un-Sus / pend"; alarm colour if $PackML$.bUn_Suspend
polyline at (260,25)-(310,35): alarm colour if $PackML$.bUn_Hold
rectangle at (260,15)-(311,31): text "Un-Hold"; alarm colour if $PackML$.bUn_Hold
polyline at (410,105)-(460,115): alarm colour if $PackML$.bComplete
rectangle at (410,95)-(461,111): text "Complete"; alarm colour if $PackML$.bComplete
polyline at (560,105)-(610,115): alarm colour if $PackML$.bSC
rectangle at (565,95)-(596,111): text "SC"; alarm colour if $PackML$.bSC
polyline at (45,130)-(55,170): alarm colour if $PackML$.bSC
rectangle at (45,140)-(76,156): text "SC"; alarm colour if $PackML$.bSC
polyline at (50,130)-(670,225): alarm colour if $PackML$.bReset OR $PackML$.Ack_Completed
rectangle at (515,210)-(576,226): text "Reset OR"; alarm colour if $PackML$.bReset
rectangle at (575,210)-(671,226): text "Ack Completed"; alarm colour if $PackML$.bAck_Completed
rectangle at (10,10)-(121,51): text "PackML / state model"
2 more shapes without text or variables
*)

(* Visualisation Simulator/MachineComponents/VC_Panel_MachineControl
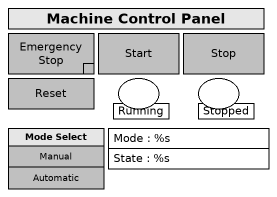
rounded rectangle at (0,25)-(86,66): text "Emergency / Stop"; alarm colour if PRG_Simulator.bBtn_EmergencyStop; toggles PRG_Simulator.bBtn_EmergencyStop
rounded rectangle at (90,25)-(171,66): text "Start"; alarm colour if .I_Btn_Start; taps .I_Btn_Start
rounded rectangle at (0,70)-(86,101): text "Reset"; alarm colour if .I_Btn_Reset; taps .I_Btn_Reset
rounded rectangle at (175,25)-(256,66): text "Stop"; alarm colour if .I_Btn_Stop; taps .I_Btn_Stop
rectangle at (0,0)-(256,21): text "Machine Control Panel"
rectangle at (100,120)-(261,141): text "Mode : %s"; shows .fbStateModel.eMode
rectangle at (100,140)-(261,161): text "State : %s"; shows .fbStateModel.eState
embedded screen at (0,120)-(96,181): VC_Panel_ModeSelector
rectangle at (105,95)-(161,111): text "Running"
rectangle at (190,95)-(246,111): text "Stopped"
ellipse at (110,70)-(151,101): alarm colour if .O_Light_Start
ellipse at (190,70)-(231,101): alarm colour if .O_Light_Stop
embedded screen at (75,55)-(86,66): VC_sensor
*)

(* Visualisation Simulator/MachineComponents/VC_Panel_ModeSelector
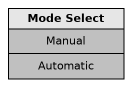
rounded rectangle at (0,20)-(116,46): text "Manual"; alarm colour if .HMI_uModeReq=3; runs INTERN ASSIGN HMI_uModeReq:=(3)
rectangle at (0,0)-(116,21): text "Mode Select"
rounded rectangle at (0,45)-(116,71): text "Automatic"; alarm colour if .HMI_uModeReq=1; runs INTERN ASSIGN HMI_uModeReq:=(1)
*)

(* Visualisation Simulator/Components/VC_Part
rectangle at (0,0)-(41,51): invisible if NOT $part$.bExists
rectangle at (15,0)-(26,41): invisible if NOT $part$.bExists OR NOT $part$.bHasHole
*)

(* Visualisation Simulator/Components/VC_sensor
rectangle at (0,0)-(11,11): alarm colour if $VAR$
*)

(* Visualisation Simulator/MachineComponents/VC_Simu_Conv_In
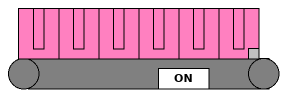
embedded screen at (210,0)-(251,51): VC_Part
embedded screen at (240,40)-(251,51): VC_sensor
embedded screen at (170,0)-(211,51): VC_Part
embedded screen at (130,0)-(171,51): VC_Part
embedded screen at (90,0)-(131,51): VC_Part
embedded screen at (50,0)-(91,51): VC_Part
embedded screen at (10,0)-(51,51): VC_Part
rectangle at (150,60)-(201,81): text "OFF"
rectangle at (150,60)-(201,81): text "ON"; invisible if NOT $MotOn$
3 more shapes without text or variables
*)

(* Visualisation Simulator/MachineComponents/VC_Simu_Drill
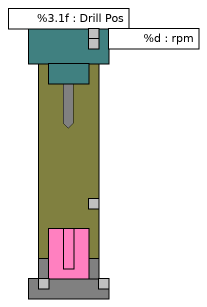
rectangle at (20,20)-(101,56): y offset $FB$.fBasePos_Y
rectangle at (0,0)-(121,21): text "%3.1f : Drill Pos"; shows $FB$.fLift_CurrentPos
embedded screen at (80,20)-(91,31): VC_sensor
embedded screen at (80,190)-(91,201): VC_sensor
embedded screen at (80,30)-(91,41): VC_sensor
polygon at (55,75)-(65,120): alarm colour if $FB$.iRPMCurrent > 0; y offset $FB$.fBasePos_Y
rectangle at (40,55)-(81,76): y offset $FB$.fBasePos_Y
rectangle at (30,250)-(41,271): x offset - $FB$.fPosJawDiff
rectangle at (80,250)-(91,271): x offset $FB$.fPosJawDiff
embedded screen at (40,220)-(81,271): VC_Part
embedded screen at (90,270)-(101,281): VC_sensor
embedded screen at (30,270)-(41,281): VC_sensor
rectangle at (100,20)-(191,41): text "%d : rpm"; shows $FB$.iRPMCurrent
2 more shapes without text or variables
*)

(* Visualisation Simulator/MachineComponents/VC_Simu_Manipulator
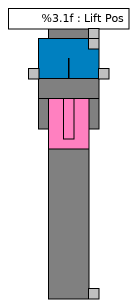
rectangle at (70,40)-(131,81): y offset $FB$.fBasePos_Y
rectangle at (100,60)-(101,81): left $FB$.fPos_Beam_L; right $FB$.fPos_Beam_R; y offset $FB$.fBasePos_Y
rectangle at (70,80)-(131,101): x offset $FB$.fPos_X; y offset $FB$.fBasePos_Y
rectangle at (70,100)-(81,131): x offset $FB$.fPos_X - $FB$.fPosFingerDiff; y offset $FB$.fBasePos_Y
rectangle at (120,100)-(131,131): x offset $FB$.fPos_X + $FB$.fPosFingerDiff; y offset $FB$.fBasePos_Y
embedded screen at (80,100)-(121,151): VC_Part
rectangle at (40,10)-(161,31): text "%3.1f : Lift Pos"; shows $FB$.fLift_CurrentPos
embedded screen at (120,30)-(131,41): VC_sensor
embedded screen at (120,290)-(131,301): VC_sensor
embedded screen at (120,40)-(131,51): VC_sensor
embedded screen at (130,70)-(141,81): VC_sensor
embedded screen at (60,70)-(71,81): VC_sensor
1 more shapes without text or variables
*)

(* Visualisation Simulator/MachineComponents/VC_SimuMach_Controls
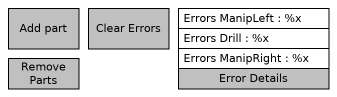
rounded rectangle at (0,0)-(71,41): text "Add part"; alarm colour if PRG_Simulator.bAddPartOnConvIn; taps PRG_Simulator.bAddPartOnConvIn
rounded rectangle at (80,0)-(161,41): text "Clear Errors"; alarm colour if PRG_Simulator.bClearErrors; taps PRG_Simulator.bClearErrors
rectangle at (170,0)-(321,21): text "Errors ManipLeft : %x"; shows PRG_Simulator.wError_ManipL; alarm colour if PRG_Simulator.wError_ManipL > 0
rounded rectangle at (0,50)-(71,81): text "Remove / Parts"; alarm colour if PRG_Simulator.bClearSystem; taps PRG_Simulator.bClearSystem
rectangle at (170,20)-(321,41): text "Errors Drill : %x"; shows PRG_Simulator.wError_Drill; alarm colour if PRG_Simulator.wError_Drill > 0
rectangle at (170,40)-(321,61): text "Errors ManipRight : %x"; shows PRG_Simulator.wError_ManipR; alarm colour if PRG_Simulator.wError_ManipR > 0
rounded rectangle at (170,60)-(321,81): text "Error Details"; opens VC_ErrorDetails
*)

(* Visualisation Simulator/VISU_SimulatedMachine
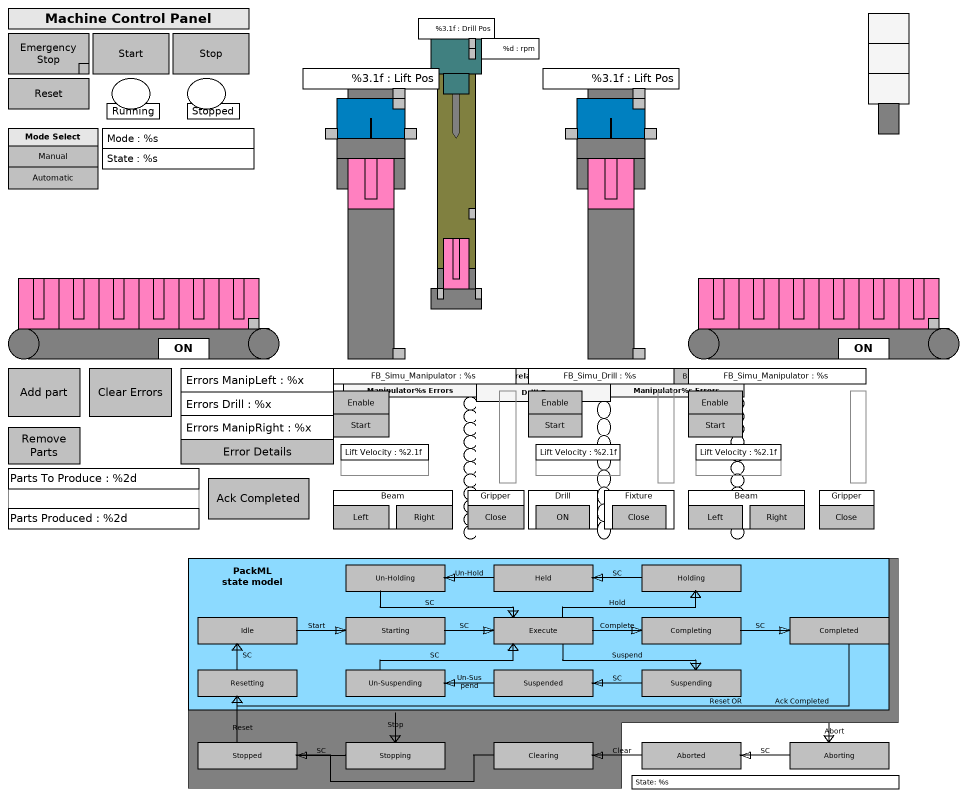
embedded screen at (335,320)-(736,491): VC_ErrorDetails
embedded screen at (0,-40)-(246,141): VC_Panel_MachineControl
embedded screen at (410,-30)-(531,261): VC_Simu_Drill
embedded screen at (0,230)-(271,311): VC_Simu_Conv_In
embedded screen at (0,320)-(326,416): VC_SimuMach_Controls
embedded screen at (325,320)-(516,481): VC_FB_Simu_Manipulator
embedded screen at (250,10)-(431,311): VC_Simu_Manipulator
embedded screen at (490,10)-(671,311): VC_Simu_Manipulator
embedded screen at (680,320)-(866,481): VC_FB_Simu_Manipulator
embedded screen at (520,320)-(666,481): VC_FB_Simu_Drill
embedded screen at (680,230)-(951,311): VC_Simu_Conv_In
embedded screen at (860,-35)-(901,86): VC_Beacon
embedded screen at (180,510)-(891,741): VC_PackMLStates
rectangle at (0,420)-(191,441): text "Parts To Produce : %2d"; shows .itemToProduce
rectangle at (0,460)-(191,481): text "Parts Produced : %2d"; shows PRG_Producing1.itemProduced
rounded rectangle at (200,430)-(301,471): text "Ack Completed"; alarm colour if .I_Btn_Start; taps .I_Btn_Ack_Completed
1 more shapes without text or variables
*)
